(* Logix 5000 project; controller SemaforoEjemplo Emulate 5570 rev 33.11; software revision 33.00 *)

TASK MainTask (continuous, watchdog 500 ms) : MainProgram

MODULES
   Local : Emulate 5570 (ICP 2, rev 33.11)
      HOLA : vendor 1 type 0 code 15 (ICP 3, rev 1.1, Output RPI 5 ms)
           Local:3:O.Data[0].0   // LUZ VERDE
           Local:3:O.Data[0].1   // LUZ AMARILLA
           Local:3:O.Data[0].2   // LUZ ROJA
END_MODULES

PROGRAM MainProgram   (* main routine MainRoutine *)
VAR
   HMI_Amarillo : BOOL;
   HMI_Rojo : BOOL;
   HMI_Verde : BOOL;
   LuzAmarilla : BOOL := 1;
   LuzRoja : BOOL;
   LuzVerde : BOOL;
   Manual : DINT;
   Manual_Automatico : BOOL;   // 1 = Manual 2 = Automatico
   Timmer : TIMER[5] := ([0].PRE := 13000, [0].ACC := 5230, [0].EN := 1, [0].TT := 1);
END_VAR

ROUTINE Automatic   (* ladder *)
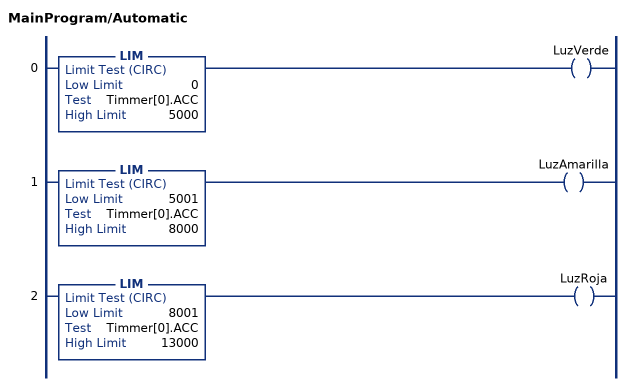
   0: LIM(0,Timmer[0].ACC,5000)OTE(LuzVerde);
   1: LIM(5001,Timmer[0].ACC,8000)OTE(LuzAmarilla);
   2: LIM(8001,Timmer[0].ACC,13000)OTE(LuzRoja);
END_ROUTINE

ROUTINE MainRoutine   (* ladder *)
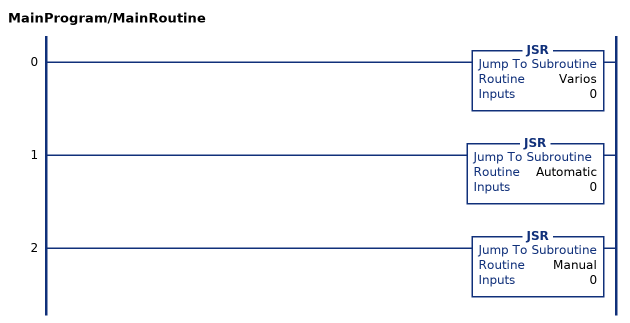
   0: JSR(Varios,0);
   1: JSR(Automatic,0);
   2: JSR(Manual,0);
END_ROUTINE

ROUTINE Manual   (* ladder *)
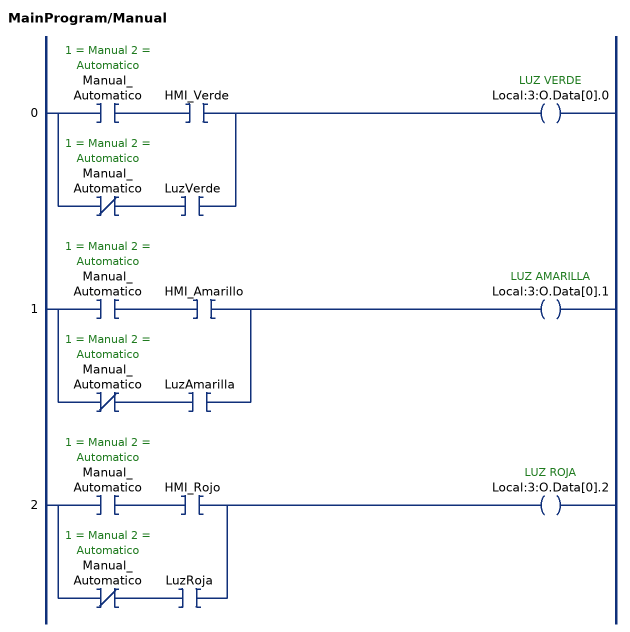
   0: [XIC(Manual_Automatico) XIC(HMI_Verde) ,XIO(Manual_Automatico) XIC(LuzVerde) ]OTE(Local:3:O.Data[0].0);
   1: [XIC(Manual_Automatico) XIC(HMI_Amarillo) ,XIO(Manual_Automatico) XIC(LuzAmarilla) ]OTE(Local:3:O.Data[0].1);
   2: [XIC(Manual_Automatico) XIC(HMI_Rojo) ,XIO(Manual_Automatico) XIC(LuzRoja) ]OTE(Local:3:O.Data[0].2);
END_ROUTINE

ROUTINE Varios   (* ladder *)
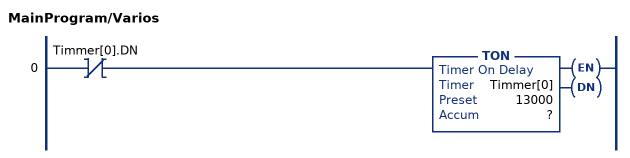
   0: XIO(Timmer[0].DN)TON(Timmer[0],?,?);
END_ROUTINE
END_PROGRAM
